FUNCTION_BLOCK FB_PDFMaker
VAR_INPUT
	
	aDataHistory			: ARRAY[0..200] OF ST_EventsHistory;
	bWriteData				: BOOL;
	aDataHistoryArrayLength	: DINT;
	nDataHistoryIndex		: DINT;
	sDate					: STRING(255);
	
	sUser					: STRING(255);
	sGroup					: STRING(255);
	sMachineName			: STRING(255);
	
	 
END_VAR
VAR_OUTPUT
	
	stJavasCriptPDF		: ST_JavasCriptPDF;
	bDataWrited			: BOOL;

END_VAR
VAR
	
	rWriteData				: R_TRIG;
	i						: DINT;
	nRowIndex				: DINT;
	sPDFDate				: STRING(255);
	bWritePDF				: BOOL;
	sFileName				: STRING(255);
	tonResetData			: TON;
	
END_VAR

ACTION ACT_IO:
stJavasCriptPDF.stEventsPdfConstants.sGroup			:= sGroup;		
stJavasCriptPDF.stEventsPdfConstants.sMachineName	:= sMachineName;
stJavasCriptPDF.stEventsPdfConstants.sUser			:= sUser;
stJavasCriptPDF.stEventsPdfConstants.sFileName		:= sFileName;
END_ACTION

ACTION ACT_WriteData:
rWriteData( CLK := bWriteData);

IF rWriteData.Q THEN
	
	FOR i := 0 TO aDataHistoryArrayLength DO
				
					stJavasCriptPDF.stEventsPDF[nRowIndex + i].sEvents					:= 	aDataHistory[i].sEventTex;
					stJavasCriptPDF.stEventsPDF[nRowIndex + i].sType					:= 	aDataHistory[i].sType;
					stJavasCriptPDF.stEventsPDF[nRowIndex + i].sDate					:= 	aDataHistory[i].sDate;
					stJavasCriptPDF.stEventsPDF[nRowIndex + i].sTime					:= 	aDataHistory[i].sTime;
				
	END_FOR
	
	i													:= 0;
	
	bDataWrited											:= TRUE;
	nRowIndex											:= nRowIndex + 201;

	

END_IF

IF nDataHistoryIndex = 0 THEN
	
	bDataWrited											:= FALSE;

END_IF

IF sPDFDate <> sDate THEN
	
	bWritePDF							:= TRUE;
	sPDFDate							:= sDate;
	
END_IF

sFileName 								:= CONCAT( STR1 := 'PDF_', STR2 := sPDFDate);

tonResetData( IN := bWritePDF, PT := T#1S);

IF tonResetData.Q THEN
	
	FOR i := 0 TO 1000 DO
				
					stJavasCriptPDF.stEventsPDF[i].sDate					:= 	'';
					stJavasCriptPDF.stEventsPDF[i].sEvents					:=  '';
					stJavasCriptPDF.stEventsPDF[i].sTime					:= 	'';
					stJavasCriptPDF.stEventsPDF[i].sType					:= 	'';
				
	END_FOR
	nRowIndex 										:= 0;		
	bWritePDF										:= FALSE;
	i												:= 0;
END_IF
END_ACTION

END_FUNCTION_BLOCK

(* stored: Version 1.1.0.1, ProductVersion 3.1.4024.13
   POU FB_PDFMaker: Id {906d47d3-6154-4696-a853-6d52290744a1}, SpecialFunc None
   Action ACT_IO: Id {8b9915ff-83a8-4047-8cda-512409519079}
   Action ACT_WriteData: Id {96624e8f-4491-4d1e-9dfe-f17cc01ba340} *)
